Staubli VAL3: ex12.pgx

program ex12()
begin
  movej(jdepart,tstylo,mlent)
  movej(ppa,tstylo,mlent)
  movel(ppb,tstylo,mlent)
  movel(ppc,tstylo,mlent)
  movej(jdepart,tstylo,mlent)
  waitEndMove()
end
